// TwinCAT 3 PLC project SetVariableFromXmlPLC
// ProgramVersion: 3.1.4024.0
// libraries:
//   Tc2_Standard, * (Beckhoff Automation GmbH)
//   Tc2_System, * (Beckhoff Automation GmbH)
//   Tc2_Utilities, * (Beckhoff Automation GmbH)
//   Tc3_DynamicMemory, * (Beckhoff Automation GmbH)
//   Tc3_JsonXml, * (Beckhoff Automation GmbH)
//   Tc3_Module, * (Beckhoff Automation GmbH)
// project tree:
//   DUTs/ ST_Device.TcDUT, ST_Variant.TcDUT
//   GVLs/ Globals.TcGVL (not stored)
//   / PlcTask.TcTTO (not stored)
//   POUs/ FB_WriteVariableByName.TcPOU, F_GetTypeFromIDS.TcPOU, MAIN.TcPOU, F_ParseToVariant.TcPOU
// real-time tasks:
//   TASK PlcTask: cycle T#1ms, priority 20, ADS port 350

// ---- DUTs/ST_Device.TcDUT
TYPE ST_Device :
STRUCT
	
	DINT_Value : DINT;
	REAL_Value : REAL; 
	BIT_Value  : BIT;

END_STRUCT
END_TYPE

// ---- DUTs/ST_Variant.TcDUT
TYPE ST_Variant :
UNION
	nBit		: BOOL;
	nI8			: SINT;
	nUI8		: USINT;
	nI16		: INT;
	nUI16		: UINT;
	nI32		: DINT;
	nUI32		: UDINT;
	nI64		: LINT;
	nUI64   : ULINT;
	fR32		: REAL;
	fR64		: LREAL;
END_UNION
END_TYPE

// ---- POUs/FB_WriteVariableByName.TcPOU
FUNCTION_BLOCK FB_WriteVariableByName

VAR_INPUT
	sName  : STRING;
	sValue : STRING;
	bExec  : BOOL;
END_VAR

VAR_OUTPUT
	Busy   : BOOL := FALSE;
	Error  : BOOL := FALSE;
	Done   :  BOOL := FALSE;
END_VAR

VAR
	nState 	: INT := 0;
	rtrig  	: R_TRIG;
	
	fbSymInfo		: PLC_ReadSymInfoByName := ( PORT := 851, TMOUT := DEFAULT_ADS_TIMEOUT );
  stSymbolInfo	: Tc2_Utilities.SYMINFOSTRUCT;
  fbWriteReq    : ADSWRITE := ( NETID := '', PORT := 851, TMOUT := DEFAULT_ADS_TIMEOUT );
	
	// Native variables for various datatypes that can be set in XML.
	// Depending on the type one variable is selected to receive the string conversion result.
  // The address will be used as data input of ADSWRITE-FB.
  
	var_data : ST_VARIANT; 
	
END_VAR

 
rtrig(CLK:= bExec , Q=> );

 CASE nState OF

	0:	// Wait for request
		IF (NOT bExec) THEN
			error := FALSE; done := FALSE;
		END_IF

		IF (rtrig.Q) THEN
			Busy:= TRUE;
			nState:= nState + 1;
		END_IF

	1:
		// reset FB
		IF (fbSymInfo.START AND NOT fbSymInfo.BUSY) THEN
			fbSymInfo( START:= FALSE);
		END_IF
		// get symbol information
		fbSymInfo
    ( 
		 	symname := sName,
	   	syminfo => stSymbolInfo,
	   	start:= TRUE
		);
		// 
		IF (NOT fbSymInfo.BUSY) THEN
	 	  IF (fbSymInfo.ERR) THEN
				nState := 99;
		  ELSE
				IF (F_ParseToVariant (adsTypeID:= stSymbolInfo.adsDataType,
							                sValue:= sValue, var_data:= var_data))
				THEN
					nState := nState + 1;
				ELSE
					nState := 99;
				END_IF
		  END_IF
		END_IF
		
	2:	// write the value
		
		// reset FB
		IF (fbWriteReq.WRITE AND NOT fbWriteReq.BUSY) THEN
			fbWriteReq(WRITE := FALSE);
		END_IF
		// write variable
		fbWriteReq
		(
			IDXGRP:= stSymbolInfo.idxGroup, 
			IDXOFFS:= stSymbolInfo.idxOffset,
			SRCADDR := ADR(var_data),
			LEN := stSymbolInfo.byteSize,
			WRITE := TRUE 
		);
		IF (NOT fbWriteReq.BUSY) THEN
	 		IF (fbWriteReq.ERR) THEN
			  nState := 99;
			ELSE
			  nState := 100;
			END_IF
		END_IF
	
	99:	// Error
		busy := FALSE;
		error := TRUE;
		nState := 0;
				
	100: // Success
		busy := FALSE;
		done := TRUE;
		nState := 0;
 
 END_CASE

END_FUNCTION_BLOCK

// ---- POUs/F_ParseToVariant.TcPOU
//
// Currently unsupported types:
//
// ADSDATATYPEID.ADST_BIGTYPE;
// ADSDATATYPEID.ADST_REAL80;
// ADSDATATYPEID.ADST_VOID;
// ADSDATATYPEID.ADST_STRING
// ADSDATATYPEID.ADST_WSTRING

FUNCTION F_ParseToVariant : bool
VAR_INPUT
	adsTypeID  : ADSDATATYPEID;
	sValue		 : STRING;
END_VAR
VAR_IN_OUT
		var_data : ST_VARIANT;
END_VAR


	F_ParseToVariant:= TRUE;	
	
	CASE adsTypeID OF 
		
		ADSDATATYPEID.ADST_INT8:
			var_data.nI8 := STRING_TO_SINT(sValue);

		ADSDATATYPEID.ADST_UINT8:
			var_data.nUI8 := STRING_TO_USINT(sValue);
					
		ADSDATATYPEID.ADST_INT16:
			var_data.nI16 := STRING_TO_INT(sValue);
		
		ADSDATATYPEID.ADST_UINT16:
			var_data.nUI16 := STRING_TO_UINT(sValue);
						
		ADSDATATYPEID.ADST_INT32:
			var_data.nI32 := STRING_TO_DINT(sValue);

		ADSDATATYPEID.ADST_UINT32:
			var_data.nUI32 := STRING_TO_UDINT(sValue);
			
		ADSDATATYPEID.ADST_INT64:
			var_data.nI64 := STRING_TO_LINT(sValue);

		ADSDATATYPEID.ADST_UINT64:
			var_data.nUI64 := STRING_TO_ULINT(sValue);			

		ADSDATATYPEID.ADST_REAL32:
			var_data.fR32 := STRING_TO_REAL(sValue);
						
		ADSDATATYPEID.ADST_REAL64:
			var_data.fR64 := STRING_TO_LREAL(sValue);
			
		ADSDATATYPEID.ADST_BIT:
			var_data.nBit := INT_TO_BOOL(STRING_TO_INT(sValue));

		ELSE
			F_ParseToVariant:= FALSE;	
		END_CASE

END_FUNCTION

// ---- POUs/F_GetTypeFromIDS.TcPOU
FUNCTION F_GetTypeFromIDS : DINT
VAR_INPUT
	ids : STRING;
END_VAR

VAR
  arIDS_ADSTypes : ARRAY[0 .. 15] OF STRING := 
	[
		'VOID',
	  'INT8',
	  'UINT8',
	  'INT16', 
    'UINT16',
		'INT32',
    'UINT32',
    'INT64',
    'UINT64',
    'REAL32',
    'REAL64',
    'BIGTYPE',
    'STRING',
    'WSTRING',
    'REAL80',
		'BIT' 
	];
										
  arID_ADSTypes  : ARRAY[0 .. 15] OF DINT := 
	[	
		ADSDATATYPEID.ADST_VOID,
		ADSDATATYPEID.ADST_INT8,
		ADSDATATYPEID.ADST_UINT8,
		ADSDATATYPEID.ADST_INT16,
		ADSDATATYPEID.ADST_UINT8,
		ADSDATATYPEID.ADST_INT32,
		ADSDATATYPEID.ADST_UINT32,
		ADSDATATYPEID.ADST_INT64,
		ADSDATATYPEID.ADST_UINT64,
		ADSDATATYPEID.ADST_REAL32,
		ADSDATATYPEID.ADST_REAL64,
		ADSDATATYPEID.ADST_BIGTYPE,
		ADSDATATYPEID.ADST_STRING,
		ADSDATATYPEID.ADST_WSTRING,
		ADSDATATYPEID.ADST_REAL80,
		ADSDATATYPEID.ADST_BIT
	];
  
	ix   : INT;
  wids : WSTRING(32);

END_VAR


F_GetTypeFromIDS := -1; // invalid

FOR ix := 0 TO 15 BY 1 DO 
 IF ids = arIDS_ADSTypes[ix] THEN 
 	F_GetTypeFromIDS:= arID_ADSTypes[ix];
	RETURN;
 END_IF; 
END_FOR; 

RETURN;

END_FUNCTION

// ---- POUs/MAIN.TcPOU
// Brief
// Reads XML string that holds initial value of variable "globals.machine.state"
// The XML is parsed and the value is applied by accessing the variable through its symbolic name.

PROGRAM MAIN
VAR
  fbXml 							: FB_XmlDomParser;
  xmlDoc 							: SXmlNode;
  xmlConfig 					: SXmlNode;
  xmlParam 						: SXmlNode;
  xmlIterator   			: SXmlIterator;
  xmlParamNode        : SXmlNode;
  xmlParamNodeValue   : STRING;
  xmlParamNodeTCType  : STRING;
  xmlParamNodeADSType : STRING;
  xmlParamNodePath    : STRING;
  
  nState 							: INT := 0;
  
  ads_type 						:  DINT;
  fbVarWriter 				: FB_WriteVariableByName;
  
  sMessageToParse : STRING(1024) := 
'<Config>
	<Parameter Path="globals.device_1.dint_value" TCType="DINT" ADSType="INT32">42</Parameter>
 	<Parameter Path="globals.device_1.real_value" TCType="REAL" ADSType="REAL32">3.1452</Parameter>
 	<Parameter Path="globals.device_2.bit_value" TCType="BIT" ADSType="BIT">1</Parameter>
</Config>';

END_VAR

CASE nState OF 
	
	0:
		(* Load XML content *)
		xmlDoc := fbXml.ParseDocument(sMessageToParse);
		xmlConfig := fbXml.ChildByName(xmlDoc, 'Config');
		xmlIterator := fbXml.Begin(xmlConfig);
		nState := nState + 1;
	
	1:	
		(* parse XML nodes *)
		IF (fbXml.IsEnd(xmlIterator)) THEN
  		xmlIterator := fbXml.End(xmlConfig);		
			nState := 100;
		ELSE
		  xmlParamNode        := fbXml.Node(xmlIterator);
  		xmlParamNodePath    :=  fbXml.AttributeText(fbXml.Attribute(n:= xmlParamNode, name:='Path'));
  		xmlParamNodeADSType := fbXml.AttributeText(fbXml.Attribute(n:= xmlParamNode, name:='ADSType'));
			xmlParamNodeValue   := fbXml.NodeText(xmlParamNode);
			// move next node
			xmlIterator := fbXml.Next(xmlIterator);
  		nState := nState + 1;
		END_IF
		
	2:	// get the variable type
	  ads_type := F_GetTypeFromIDS( xmlParamNodeADSType);
		IF (ads_type < 0) THEN // Unsupported type. For now we will end with error.
			nState := 99;
		ELSE 
			nState := nState + 1;
		END_IF
		
	3: 	
			IF (fbVarWriter.bExec AND NOT fbVarWriter.Busy) THEN
				fbVarWriter( bExec := FALSE);
			END_IF
			fbVarWriter
			(
				bExec  := TRUE,
				sName  := xmlParamNodePath,
				sValue := xmlParamNodeValue
			);
			IF (NOT fbVarWriter.Busy) THEN
				IF (fbVarWriter.Error) THEN
					;
				END_IF
				fbVarWriter( bExec := FALSE);
				nState := 1;
			END_IF
		
	99:	 // Error
	
	100: // Finished

END_CASE

END_PROGRAM
